{attribute 'qualified_only'}
VAR_GLOBAL
 PlcToPc: ARRAY[0..1023] OF BYTE;
END_VAR

(* stored: Version 1.1.0.1, ProductVersion 3.1.4024.5
   GVL _PlcToPc: Id {3de8834f-3a2e-4ef1-945e-9d80ea855cd2} *)
